FUNCTION Get_Bool_From_Buffer : Buffer_Error
VAR_INPUT
	Num : USINT;
	Layout : REFERENCE TO Buffer_Layout;
END_VAR

VAR_IN_OUT
	Buffer : ARRAY [*] OF BYTE;
	Out : BOOL;
END_VAR

VAR
	Offset : USINT;
	CopyByte : BYTE;
	P_Int : POINTER TO BOOL;
	BufferSize : DINT;
	i : UINT;
END_VAR

BufferSize := UPPER_BOUND(Buffer, 1) - LOWER_BOUND(Buffer, 1); // berekent buffer size

IF BufferSize = Layout.Buffer_Size THEN
	Get_Bool_From_Buffer := Buffer_Error.Layout_Not_Size_Buffer; // return error dat buffer size niet overeen komt met buffer layout
	RETURN;
END_IF

IF NOT Layout.Enabel_Bool_Array THEN
	Get_Bool_From_Buffer := Buffer_Error.Array_Not_Enabelt; // return error data array niet enabelt is
	RETURN;
END_IF

IF Num > Layout.Bool_Amount THEN
	Get_Bool_From_Buffer := Buffer_Error.Array_To_Small; // return error data de num niet in de type array past
	RETURN;
END_IF

Offset := Layout.Bool_Array_Offset + (Num * 1);

IF Offset > BufferSize THEN // chek of float in buffer past met offset
	Out := FALSE; // return
	Get_Bool_From_Buffer := Buffer_Error.Read_Error; // return error read out of bouds van arry
	RETURN;
ELSE
	CopyByte := Buffer[Offset];
	P_Int := ADR(CopyByte); // maak een pinter van de buffer
	Get_Bool_From_Buffer := Buffer_Error.None;
	Out := P_Int^; // return
END_IF

END_FUNCTION

(* stored: Version 1.1.0.1, ProductVersion 3.1.4024.10
   POU Get_Bool_From_Buffer: Id {b573418b-f7a5-4a55-9649-f2f572babd57}, SpecialFunc None *)
